// TIA Portal V18 export
FUNCTION_BLOCK "Sequencer"   // FB4, GRAPH
VERSION : 0.1
// stored: AcknowledgeErrorsRequired true, AutoNumber true, ExtensionBlockName "ExtensionToGRAPH", GraphVersion 5.0, InitialValuesAcquisition true, IsIECCheckEnabled true, LanguageInNetworks FBD, LockOperatingMode false, PermanentILProcessingInMANMode false, SetENOAutomatically false, SkipSteps false, UDAEnableTagReadback false, WithAlarmHandling true
   // inherited from GRAPH_BASE
   VAR
      OFF_SQ_BASE : Bool;
   END_VAR
   VAR_INPUT
      OFF_SQ { ExternalWritable := 'False'} : Bool := false;   // Kette ausschalten / Turn sequence off / Désactiver le graphe
      INIT_SQ { ExternalWritable := 'False'} : Bool := false;   // Kette in Initialzustand versetzen
      ACK_EF { ExternalWritable := 'False'} : Bool := false;   // Alle Fehler und Störungen quittieren / Acknowledge all errors and faults / Acquitter toutes les erreurs et perturbations
      REG_EF { ExternalWritable := 'False'} : Bool := false;   // Alle Fehler und Störungen registrieren / Register all errors and faults / Enregistrer toutes les erreurs et perturbations
      ACK_S { ExternalWritable := 'False'} : Bool := false;   // Schritt quittieren, der an Parameter S_NO anliegt / Acknowledge step indicated in S_NO / Acquitter l'étape figurant dans le paramètre S_NO
      REG_S { ExternalWritable := 'False'} : Bool := false;   // Schritt registrieren, der an Parameter S_NO anliegt / Register the step indicated in S_NO / Enregistrer l'étape figurant dans le paramètre S_NO
      HALT_SQ { ExternalWritable := 'False'} : Bool := false;   // Kette sofort anhalten / Halt sequence immediately / Arrêter le graphe immédiatement
      HALT_TM { ExternalWritable := 'False'} : Bool := false;   // Zeiten sofort anhalten / Halt timers immediately / Arrêter les temporisations immédiatement
      ZERO_OP { ExternalWritable := 'False'} : Bool := false;   // Alle mit N, L, D zugewiesenen Operanden auf 0 setzen / Set all operands assigned with N, L, D to 0 / Mettre à 0 tous les opérandes affectés avec N, L, D
      EN_IL { ExternalWritable := 'False'} : Bool := false;   // Interlockbearbeitung aktivieren / Activate interlocks / Activer le traitement des Interlocks
      EN_SV { ExternalWritable := 'False'} : Bool := false;   // Supervisionsbearbeitung aktivieren / Activate supervision processing / Activer le traitement de Supervision
      EN_ACKREQ { ExternalWritable := 'False'} : Bool := false;   // Quittierpflicht aktivieren / Activate mandatory acknowledgment / Activer l'obligation d'acquittement
      EN_SSKIP { ExternalWritable := 'False'} : Bool := false;   // "Schritte überspringen" aktivieren / Enable "Skip step" / Activer "Ignorer l'étape"
      DISP_SACT { ExternalWritable := 'False'} : Bool := false;   // Nur aktive Schritte anzeigen / Display active steps only / Afficher uniquement les étapes activées
      DISP_SEF { ExternalWritable := 'False'} : Bool := false;   // Nur fehlerhafte und gestörte Schritte anzeigen / Display only steps with errors and disrupted steps / Afficher uniquement les étapes avec erreurs et perturbations
      DISP_SALL { ExternalWritable := 'False'} : Bool := false;   // Alle Schritte anzeigen / Display all steps / Afficher toutes les étapes
      S_PREV { ExternalWritable := 'False'} : Bool := false;   // Vorherigen Schritt am Parameter S_NO ausgeben / Output previous step in parameter S_NO / Afficher l'étape précédente dans le paramètre S_NO
      S_NEXT { ExternalWritable := 'False'} : Bool := false;   // Nächsten Schritt am Parameter S_NO anzeigen / Indicate next step in parameter S_NO / Afficher l'étape suivante dans le paramètre S_NO
      SW_AUTO { ExternalWritable := 'False'} : Bool := false;   // Automatischer Betrieb / Automatic mode / Mode automatique
      SW_TAP { ExternalWritable := 'False'} : Bool := false;   // Halbautomatisch/Weiterschalten mit Transition / Semiautomatic/switch with transition / Mode semi-automatique/Activation de l'étape suivante avec transition
      SW_TOP { ExternalWritable := 'False'} : Bool := false;   // Halbautomatisch/Ignoriere Transition / Semiautomatic/ignore transition / Mode semi-automatique/Ignorer la transition
      SW_MAN { ExternalWritable := 'False'} : Bool := false;   // Handbetrieb / Manual mode / Mode manuel
      S_SEL { ExternalWritable := 'False'} : Int := 0;   // Schritt auswählen, der an S_NO ausgegeben werden soll / Select step to be output to S_NO / Sélectionner l'étape à afficher dans S_NO
      S_SELOK { ExternalWritable := 'False'} : Bool := false;   // Wert aus S_SEL nach S_NO übernehmen / Enter value from S_SEL in S_NO / Appliquer la valeur de S_SEL à S_NO
      S_ON { ExternalWritable := 'False'} : Bool := false;   // Schritt aktivieren, der an Parameter S_NO anliegt / Activate step indicated in S_NO / Activer l'étape figurant dans le paramètre S_NO
      S_OFF { ExternalWritable := 'False'} : Bool := false;   // Schritt deaktivieren, der an Parameter S_NO anliegt / Deactivate step indicated S_NO / Désactiver l'étape figurant dans le paramètre S_NO
      T_PREV { ExternalWritable := 'False'} : Bool := false;   // Vorherige Transition an Parameter T_NO anzeigen / Display previous transition in T_NO / Afficher la transition précédente dans le paramètre T_NO
      T_NEXT { ExternalWritable := 'False'} : Bool := false;   // Nächste Transition an Parameter T_NO anzeigen / Display next transition at parameter T_NO / Afficher la transition suivante dans le paramètre T_NO
      T_PUSH { ExternalWritable := 'False'} : Bool := false;   // Schaltfreigabe für Transition im halbautomatischen Betrieb / Enable transition to switch in semi automatic mode / Validation de commutation pour transition en mode semi-automatique
      EN_LMODE { ExternalWritable := 'False'} : Bool := false;   // Lernmodus aktivieren / Activate learning mode / Activer le mode apprentissage
      RESET_CRIT { ExternalWritable := 'False'} : Bool := false;   // Alle Erstwerte, die für Interlocks und Transitionen aufgezeichnet wurden, zurücksetzen / Reset all initial values recorded for interlocks and transitions / Réinitialiser toutes les premières valeurs enregistrées pour les Interlocks et les transitions
      startButton : Bool;
      lightBeam1 : Bool;
      lightBeam2 : Bool;
      lightBeam3 : Bool;
      robotArmDown : Bool;
      robotOnStation : Bool;
      robotOnMagazine : Bool;
      mySupervision : Bool;
   END_VAR
   VAR_OUTPUT
      S_NO { ExternalWritable := 'False'} : Int := 0;   // Schrittnummer / Step number / Numéro d'étape
      S_MORE { ExternalWritable := 'False'} : Bool := false;   // Weitere Schritte sind vorhanden und können in S_NO angezeigt werden. / More steps are available and can be shown in S_NO / Il existe d'autres étapes qui peuvent être affichées dans S_NO.
      S_ACTIVE { ExternalWritable := 'False'} : Bool := false;   // Schritt, der an Parameter S_NO angezeigt wird, ist aktiv / Step indicated in S_NO is active / L'étape affichée dans le paramètre S_NO est activée
      S_TIME { ExternalWritable := 'False'} : Time := T#0ms;   // Schrittaktivierungszeit / Step activation time / Temps d'activation d'étape
      S_TIMEOK { ExternalWritable := 'False'} : Time := T#0ms;   // Schrittaktivierungszeit fehlerfrei / No error in step activation time / Temps d'activation d'étape sans erreur
      S_CRITLOC { ExternalWritable := 'False'} : DWord := 16#0;   // Interlock-Kriterienbits / Interlock criteria bits / Bits de critère Interlock
      S_CRITLOCERR { ExternalWritable := 'False'} : DWord := 16#0;   // Interlock-Kriterienbits bei Ereignis L1 / Interlock criteria bits for event L1 / Bits de critère Interlock pour l'événement L1
      S_STATE { ExternalWritable := 'False'} : Word := 16#0;   // Schrittzustandsbits / Step state bits / Bits d'état d'étape
      T_NO { ExternalWritable := 'False'} : Int := 0;   // Transitionsnummer / Transition number / Numéro de transition
      T_MORE { ExternalWritable := 'False'} : Bool := false;   // Weitere gültige Transitionen zur Anzeige verfügbar / More valid transitions available for display / D'autres transitions valides sont disponibles pour affichage
      T_CRIT { ExternalWritable := 'False'} : DWord := 16#0;   // Transitions-Kriterienbits / Transition criteria bits / Bits de critère de transition
      T_CRITOLD { ExternalWritable := 'False'} : DWord := 16#0;   // Transitions-Kriterienbits des letzten Zyklus / Transition criteria bits from last cycle / Bits de critère de transition du dernier cycle
      T_CRITFLT { ExternalWritable := 'False'} : DWord := 16#0;   // Transitions-Kriterienbits bei Ereignis V1 / Transition criteria bits for event V1 / Bits de critère de transition pour l'événement V1
      ERROR { ExternalWritable := 'False'} : Bool := false;   // Sammelfehler Interlock / Interlock group error / Erreur groupée Interlock
      FAULT { ExternalWritable := 'False'} : Bool := false;   // Sammelfehler Supervision / Supervision group error / Erreur groupée Supervision
      ERR_FLT { ExternalWritable := 'False'} : Bool := false;   // Sammelfehler Interlock oder Supervision / Interlock or supervision group error / Erreur groupée Interlock or Supervision
      SQ_ISOFF { ExternalWritable := 'False'} : Bool := false;   // Kette ausgeschaltet (kein Schritt aktiv) / Sequence is off (no step active) / Graphe désactivé (aucune étape n'est activée)
      SQ_HALTED { ExternalWritable := 'False'} : Bool := false;   // Kette angehalten / Sequence halted / Graphe arrêté
      TM_HALTED { ExternalWritable := 'False'} : Bool := false;   // Zeiten angehalten / Timers halted / Les temporisations sont arrêtées
      OP_ZEROED { ExternalWritable := 'False'} : Bool := false;   // Alle mit N, L oder D zugewiesenen Operanden auf 0 gesetzt / All the operands assigned with N, L, D are set to 0 / Tous les opérandes affectés avec N, L ou D sont mis à 0
      IL_ENABLED { ExternalWritable := 'False'} : Bool := false;   // Interlockbearbeitung aktiv / Interlocks are active / Traitement des Interlocks activé
      SV_ENABLED { ExternalWritable := 'False'} : Bool := false;   // Supervisionsbearbeitung aktiviert / Supervision processing activated / Traitement de Supervision activé
      ACKREQ_ENABLED { ExternalWritable := 'False'} : Bool := false;   // Quittierpflicht aktiviert / Mandatory acknowledgment activated / Obligation d'acquittement activée
      SSKIP_ENABLED { ExternalWritable := 'False'} : Bool := false;   // Schritte überspringen aktiviert / Skip steps activated / Ignorer les étapes activé
      SACT_DISP { ExternalWritable := 'False'} : Bool := false;   // Nur aktive Schritte anzeigen / Display active steps only / Afficher uniquement les étapes activées
      SEF_DISP { ExternalWritable := 'False'} : Bool := false;   // Nur fehlerhafte oder gestörte Schritte anzeigen / Display only steps with errors or disrupted steps / Afficher uniquement les étapes avec erreurs ou perturbations
      SALL_DISP { ExternalWritable := 'False'} : Bool := false;   // Alle Schritte anzeigen / Display all steps / Afficher toutes les étapes
      AUTO_ON { ExternalWritable := 'False'} : Bool := false;   // Automatischer Betrieb eingeschaltet / Automatic mode is active / Mode automatique activé
      TAP_ON { ExternalWritable := 'False'} : Bool := false;   // Halbautomatischer Betrieb/Schritt mit Transition eingeschaltet / Semiautomatic mode/step with transition enabled / Mode semi-automatique/Etape avec transition activé
      TOP_ON { ExternalWritable := 'False'} : Bool := false;   // Halbautomatischer Betrieb/Ignoriere Transition eingeschaltet / Semiautomatic mode/ignore transition enabled / Mode semi-automatique/Ignorer la transition activé
      MAN_ON { ExternalWritable := 'False'} : Bool := false;   // Handbetrieb eingeschaltet / Manual mode is active / Mode manuel activé
      LMODE_ENABLED { ExternalWritable := 'False'} : Bool := false;   // Lernmodus aktiv / Learning mode is active / Mode apprentissage actif
      partInPos1 : Bool;
      partInPos2 : Bool;
      partInPos3 : Bool;
      startConv : Bool;
      automaticMode : Bool;
      robotFill : Bool;
      robotGoToMagazine : Bool;
      robotGoToStation : Bool;
   END_VAR
   VAR
      safetyOK { ExternalAccessible := 'False'; ExternalVisible := 'False'; ExternalWritable := 'False'} : Bool;
      statLightbeam3Fal : Bool;
      statMemoryTag : Bool;
      instExtensionToGRAPH { S7_SetPoint := 'True'} : "ExtensionToGRAPH";
   END_VAR
   VAR_TEMP   // added for the SCL form of the ladder/FBD networks
      _w1 : Bool;
   END_VAR
BEGIN
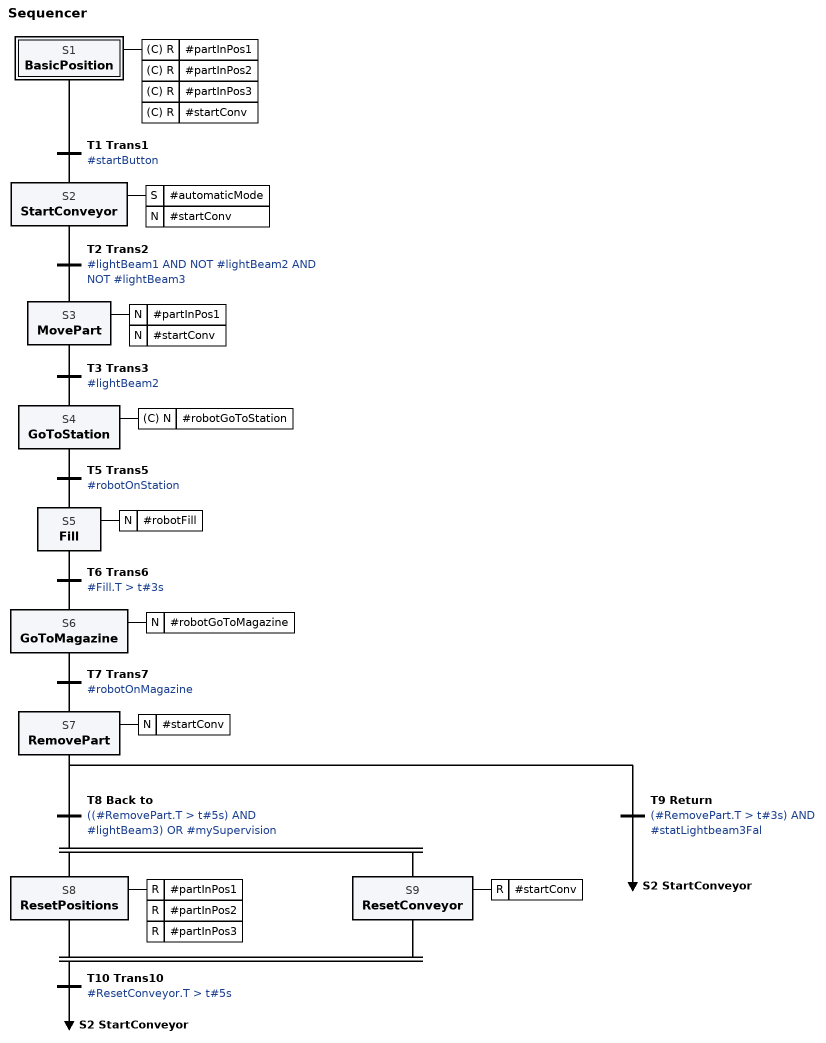
   // sequencer 1
   // //=============================================================================
   // //Siemens AG // (c)Copyright (2018)
   // //-----------------------------------------------------------------------------
   // // Library: -
   // // Tested with: CPU 1517-3 PN/DP V2.5
   // // Engineering: TIA Portal V15
   // // Restrictions: -
   // // Requirements: PLC (S7-1500)
   // // Functionality: Sequencer
   // //-----------------------------------------------------------------------------
   // // Change log table:
   // // Version    Date         Expert in charge  Changes applied
   // // 01.00.00 24.08.18  Siemens                First released version
   // //=============================================================================
   INITIAL_STEP BasicPosition:   // S1, max time T#10S, warning time T#7S
      interlock C := #safetyOK;   // Интерлок если сафети не в порядке / сообщение от интерлока / safety not OK
      supervision V := (#StartConveyor.U > t#100ms) AND (#StartConveyor.T > t#100ms);   // Suppervision =1 - fault / сообщение от супервизион / Step activation time
      (C)     R    #partInPos1
      (C)     R    #partInPos2
      (C)     R    #partInPos3
      (C)     R    #startConv
   END_STEP
   TRANSITION Trans1 FROM BasicPosition TO StartConveyor   // T1
      := #startButton;
   END_TRANSITION
   STEP StartConveyor:   // S2, max time T#10S, warning time T#7S
              S    #automaticMode
              N    #startConv
   END_STEP
   TRANSITION Trans2 FROM StartConveyor TO MovePart   // T2
      := #lightBeam1 AND NOT #lightBeam2 AND NOT #lightBeam3;
   END_TRANSITION
   STEP MovePart:   // S3, max time T#10S, warning time T#7S
      supervision V := (none);   // Schrittaktivierungszeit überschritten / Step activation time is exceeded
              N    #partInPos1
              N    #startConv
   END_STEP
   TRANSITION Trans3 FROM MovePart TO GoToStation   // T3
      := #lightBeam2;
   END_TRANSITION
   STEP GoToStation:   // S4, max time T#10S, warning time T#7S
      interlock C := NOT #robotArmDown;   // Robot is up
      (C)     N    #robotGoToStation
   END_STEP
   TRANSITION Trans5 FROM GoToStation TO Fill   // T5
      := #robotOnStation;
   END_TRANSITION
   STEP Fill:   // S5, max time T#10S, warning time T#7S
              N    #robotFill
   END_STEP
   TRANSITION Trans6 FROM Fill TO GoToMagazine   // T6
      := #Fill.T > t#3s;
   END_TRANSITION
   STEP GoToMagazine:   // S6, max time T#10S, warning time T#7S
              N    #robotGoToMagazine
   END_STEP
   TRANSITION Trans7 FROM GoToMagazine TO RemovePart   // T7
      := #robotOnMagazine;
   END_TRANSITION
   STEP RemovePart:   // S7, max time T#10S, warning time T#7S
      supervision V := (#RemovePart.T < #RemovePart.T_MAX) AND (#RemovePart.T > #RemovePart.T_WARN);   // Schrittaktivierungszeit überschritten / Step activation time is exceeded
              N    #startConv
   END_STEP
   TRANSITION "Back to" FROM RemovePart TO (ResetPositions, ResetConveyor)   // T8
      := ((#RemovePart.T > t#5s) AND #lightBeam3) OR #mySupervision;
   END_TRANSITION
   TRANSITION "Return" FROM RemovePart TO StartConveyor   // T9, jump
      := (#RemovePart.T > t#3s) AND #statLightbeam3Fal;
   END_TRANSITION
   STEP ResetPositions:   // S8, max time T#10S, warning time T#7S
      interlock C := #ResetPositions.T > #ResetPositions.T_MAX;   // Interlocks deaktivieren / Deactivate interlocks
      supervision V := (none);   // Supervision is TRUE, please set it to FALSE
              R    #partInPos1
              R    #partInPos2
              R    #partInPos3
   END_STEP
   TRANSITION Trans10 FROM (ResetConveyor, ResetPositions) TO StartConveyor   // T10, jump
      := #ResetConveyor.T > t#5s;
   END_TRANSITION
   STEP ResetConveyor:   // S9, max time T#10S, warning time T#7S
              R    #startConv
   END_STEP

   // permanent post-instructions
   NETWORK 1
      #_w1 := NOT #lightBeam3 AND #statMemoryTag;   // falling edge of #lightBeam3
      #statMemoryTag := #lightBeam3;
      #statLightbeam3Fal := #_w1;
END_FUNCTION_BLOCK
